// reads usage/free and total space of hdd
{attribute 'monitoring' := 'call'}
INTERFACE PUBLIC I_HddUsage

// LO = FB is finished -> data valid
{attribute 'monitoring' := 'call'}
PROPERTY PUBLIC Busy : BOOL
GET
END_GET
END_PROPERTY

// number of bytes free to use
{attribute 'monitoring' := 'call'}
PROPERTY PUBLIC BytesFree : ULINT
GET
END_GET
END_PROPERTY

// total capacity of hdd in bytes
{attribute 'monitoring' := 'call'}
PROPERTY PUBLIC BytesTotal : ULINT
GET
END_GET
END_PROPERTY

// number of bytes free already used
{attribute 'monitoring' := 'call'}
PROPERTY PUBLIC BytesUsed : ULINT
GET
END_GET
END_PROPERTY

// drive letter
{attribute 'monitoring' := 'call'}
PROPERTY PUBLIC Drive : STRING[2]
GET
END_GET
END_PROPERTY

// HI = unable to retrieve data
{attribute 'monitoring' := 'call'}
PROPERTY PUBLIC Error : BOOL
GET
END_GET
END_PROPERTY

// percentual free space
{attribute 'monitoring' := 'call'}
PROPERTY PUBLIC PercentageFree : BYTE
GET
END_GET
END_PROPERTY

// percentual used space
{attribute 'monitoring' := 'call'}
PROPERTY PUBLIC PercentageUsed : BYTE
GET
END_GET
END_PROPERTY

END_INTERFACE

(* stored: Version 1.1.0.1, ProductVersion 3.1.4024.4
   Itf I_HddUsage: Id {98b5570c-fa8a-41b0-8781-84655e04dabb}
   Folder properties: Id {12f23bd7-155f-4d7a-b639-f7822868fe1c}
   Property Busy: Id {6881636d-02d9-4677-b70e-6951d62c7080}
   Get Get: Id {9d0b1399-5ae9-4ebb-b8ab-f87c986dad2a}
   Property BytesFree: Id {2685f038-065a-4131-86de-1abe15dbeca1}
   Get Get: Id {ad917130-0f7a-4d6d-b118-bf600bd74f99}
   Property BytesTotal: Id {b1fa7935-cfcc-457c-8aee-746303f33746}
   Get Get: Id {ad040f8a-337c-45fc-986b-affe0310600d}
   Property BytesUsed: Id {b2b05c58-b084-48c1-a334-55fb4dbf1e9f}
   Get Get: Id {75ec8fda-be0c-408f-9ead-5f17c29da86a}
   Property Drive: Id {b846b76f-1a20-428c-b729-7041e2242c06}
   Get Get: Id {86fc5f39-15d9-407f-b68f-5a72e8cb0dee}
   Property Error: Id {1524f1de-56c1-4790-97f8-2c092010b73c}
   Get Get: Id {32d32e52-7e5e-45a3-80b7-dca5315dd40f}
   Property PercentageFree: Id {3126a29b-33ab-4f1b-b61a-3ebeb3b0f8e2}
   Get Get: Id {2705e4e0-0fde-44d4-9799-32de5784d5d1}
   Property PercentageUsed: Id {935c460e-f77e-4082-bd7c-a63113d07eaf}
   Get Get: Id {c203c7ac-1e5b-4d87-8836-b9540aa8a5f9} *)
